// TIA Portal project "Ejercicio2_AutoGarbigailua" (V15.1)

(* hardware
DEVICE "S7-1200 station_1"  S7-1200 Station
   slot 0: "Rack_0"  S7-1200 Rack  Rack  V1.0
   slot 1: "PLC_1"  CPU 1214C AC/DC/Rly  6ES7 214-1BG40-0XB0  V4.2
*)

// ===== PLC "PLC_1"  CPU 1214C AC/DC/Rly =====

VAR_GLOBAL   // PLC tag table "Tabla de variables estándar"
   "Etapa4" AT %M16.4 : Bool;
   "Etapa3" AT %M16.3 : Bool;
   "Etapa2" AT %M16.2 : Bool;
   "Etapa1" AT %M16.1 : Bool;
   "Etapa0" AT %M16.0 : Bool;
   "S1" AT %I1.0 : Bool;
   "S2" AT %I1.1 : Bool;
   "S3" AT %I1.2 : Bool;
   "M" AT %I1.3 : Bool;
   "P" AT %I1.4 : Bool;
   "XV" AT %Q1.0 : Bool;
   "MP" AT %Q1.1 : Bool;
   "MC" AT %Q1.2 : Bool;
   "MV" AT %Q1.3 : Bool;
   "Etapa1.1" AT %M1.0 : Bool;
   "Etapa2.1" AT %M1.1 : Bool;
   "Etapa3.1" AT %M1.2 : Bool;
   "Etapa4.1" AT %M1.3 : Bool;
END_VAR

ORGANIZATION_BLOCK "Main"   // OB1, LAD, ProgramCycle
TITLE = "Main Program Sweep (Cycle)"
{ S7_Optimized_Access := 'TRUE' }
VERSION : 0.1
   VAR_INPUT
      Initial_Call : Bool;   // Initial call of this OB
      Remanence : Bool;   // =True, if remanent data are available
   END_VAR
   VAR_TEMP   // added for the SCL form of the ladder/FBD networks
      _w1 : Bool;
   END_VAR
BEGIN

REGION Network 1
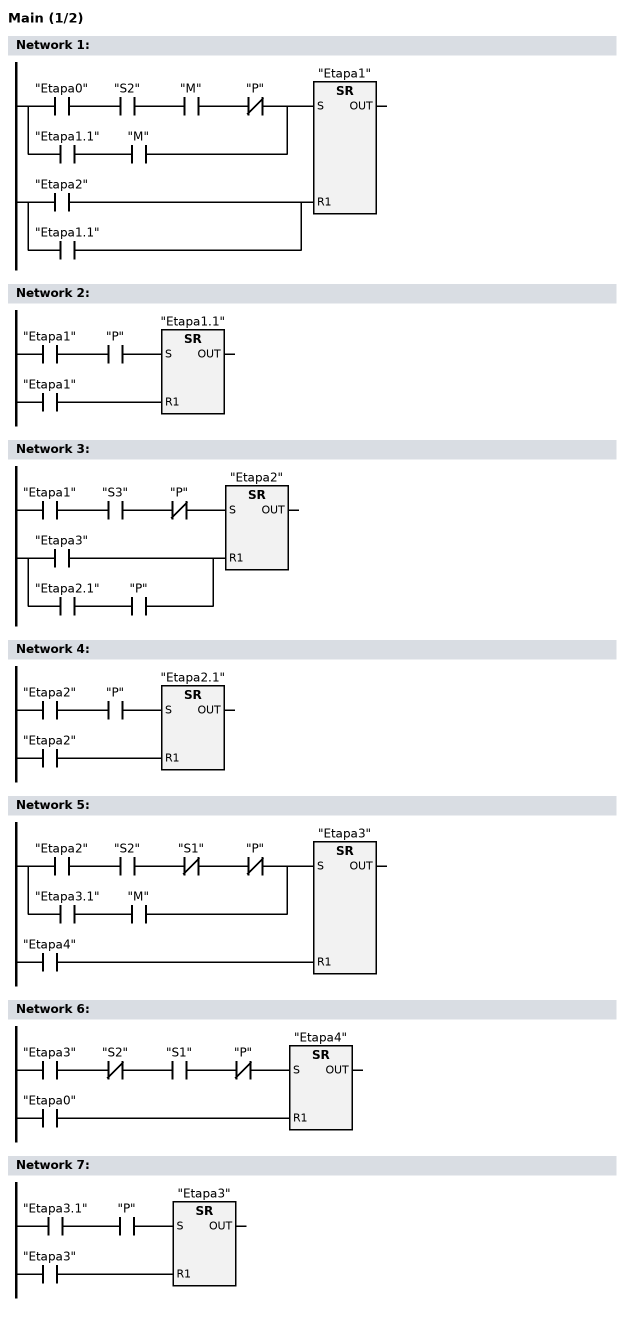
   RUNG wire#powerrail
      Contact( "Etapa0" )
      Contact( "S2" )
      Contact( "M" )
      I_Contact( "P" )
      wire#w1
      S_SR(operand := "Etapa1", r1 := wire#w2)
   END_RUNG
   RUNG wire#powerrail
      Contact( "Etapa1.1" )
      Contact( "M" )
   END_RUNG wire#w1
   RUNG wire#powerrail
      Contact( "Etapa2" )
   END_RUNG wire#w2
   RUNG wire#powerrail
      Contact( "Etapa1.1" )
   END_RUNG wire#w2
   // the same network as SCL:
   IF ("Etapa0" AND "S2" AND "M" AND NOT "P") OR ("Etapa1.1" AND "M") THEN
       "Etapa1" := TRUE;   // SR flip-flop
   END_IF;
   IF "Etapa2" OR "Etapa1.1" THEN "Etapa1" := FALSE; END_IF;
END_REGION

REGION Network 2
   RUNG wire#powerrail
      Contact( "Etapa1" )
      Contact( "P" )
      S_SR(operand := "Etapa1.1", r1 := wire#w1)
   END_RUNG
   RUNG wire#powerrail
      Contact( "Etapa1" )
   END_RUNG wire#w1
   // the same network as SCL:
   IF "Etapa1" AND "P" THEN
       "Etapa1.1" := TRUE;   // SR flip-flop
   END_IF;
   IF "Etapa1" THEN "Etapa1.1" := FALSE; END_IF;
END_REGION

REGION Network 3
   RUNG wire#powerrail
      Contact( "Etapa1" )
      Contact( "S3" )
      I_Contact( "P" )
      S_SR(operand := "Etapa2", r1 := wire#w1)
   END_RUNG
   RUNG wire#powerrail
      Contact( "Etapa3" )
   END_RUNG wire#w1
   RUNG wire#powerrail
      Contact( "Etapa2.1" )
      Contact( "P" )
   END_RUNG wire#w1
   // the same network as SCL:
   IF "Etapa1" AND "S3" AND NOT "P" THEN
       "Etapa2" := TRUE;   // SR flip-flop
   END_IF;
   IF "Etapa3" OR ("Etapa2.1" AND "P") THEN "Etapa2" := FALSE; END_IF;
END_REGION

REGION Network 4
   RUNG wire#powerrail
      Contact( "Etapa2" )
      Contact( "P" )
      S_SR(operand := "Etapa2.1", r1 := wire#w1)
   END_RUNG
   RUNG wire#powerrail
      Contact( "Etapa2" )
   END_RUNG wire#w1
   // the same network as SCL:
   IF "Etapa2" AND "P" THEN
       "Etapa2.1" := TRUE;   // SR flip-flop
   END_IF;
   IF "Etapa2" THEN "Etapa2.1" := FALSE; END_IF;
END_REGION

REGION Network 5
   RUNG wire#powerrail
      Contact( "Etapa2" )
      Contact( "S2" )
      I_Contact( "S1" )
      I_Contact( "P" )
      wire#w1
      S_SR(operand := "Etapa3", r1 := wire#w2)
   END_RUNG
   RUNG wire#powerrail
      Contact( "Etapa3.1" )
      Contact( "M" )
   END_RUNG wire#w1
   RUNG wire#powerrail
      Contact( "Etapa4" )
   END_RUNG wire#w2
   // the same network as SCL:
   IF ("Etapa2" AND "S2" AND NOT "S1" AND NOT "P") OR ("Etapa3.1" AND "M") THEN
       "Etapa3" := TRUE;   // SR flip-flop
   END_IF;
   IF "Etapa4" THEN "Etapa3" := FALSE; END_IF;
END_REGION

REGION Network 6
   RUNG wire#powerrail
      Contact( "Etapa3" )
      I_Contact( "S2" )
      Contact( "S1" )
      I_Contact( "P" )
      S_SR(operand := "Etapa4", r1 := wire#w1)
   END_RUNG
   RUNG wire#powerrail
      Contact( "Etapa0" )
   END_RUNG wire#w1
   // the same network as SCL:
   IF "Etapa3" AND NOT "S2" AND "S1" AND NOT "P" THEN
       "Etapa4" := TRUE;   // SR flip-flop
   END_IF;
   IF "Etapa0" THEN "Etapa4" := FALSE; END_IF;
END_REGION

REGION Network 7
   RUNG wire#powerrail
      Contact( "Etapa3.1" )
      Contact( "P" )
      S_SR(operand := "Etapa3", r1 := wire#w1)
   END_RUNG
   RUNG wire#powerrail
      Contact( "Etapa3" )
   END_RUNG wire#w1
   // the same network as SCL:
   #_w1 := "Etapa3";
   IF "Etapa3.1" AND "P" THEN
       "Etapa3" := TRUE;   // SR flip-flop
   END_IF;
   IF #_w1 THEN "Etapa3" := FALSE; END_IF;
END_REGION

REGION Network 8
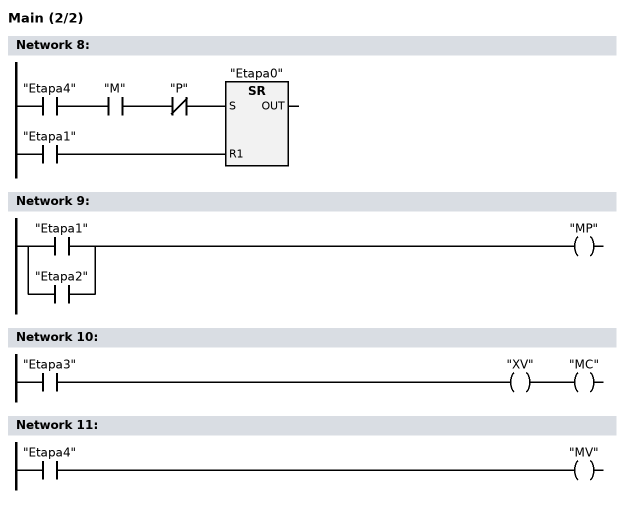
   RUNG wire#powerrail
      Contact( "Etapa4" )
      Contact( "M" )
      I_Contact( "P" )
      S_SR(operand := "Etapa0", r1 := wire#w1)
   END_RUNG
   RUNG wire#powerrail
      Contact( "Etapa1" )
   END_RUNG wire#w1
   // the same network as SCL:
   IF "Etapa4" AND "M" AND NOT "P" THEN
       "Etapa0" := TRUE;   // SR flip-flop
   END_IF;
   IF "Etapa1" THEN "Etapa0" := FALSE; END_IF;
END_REGION

REGION Network 9
   RUNG wire#powerrail
      Contact( "Etapa1" )
      wire#w1
      Coil( "MP" )
   END_RUNG
   RUNG wire#powerrail
      Contact( "Etapa2" )
   END_RUNG wire#w1
   // the same network as SCL:
   "MP" := "Etapa1" OR "Etapa2";
END_REGION

REGION Network 10
   RUNG wire#powerrail
      Contact( "Etapa3" )
      Coil( "XV" )
      Coil( "MC" )
   END_RUNG
   // the same network as SCL:
   "XV" := "Etapa3";
   "MC" := "Etapa3";
END_REGION

REGION Network 11
   RUNG wire#powerrail
      Contact( "Etapa4" )
      Coil( "MV" )
   END_RUNG
   // the same network as SCL:
   "MV" := "Etapa4";
END_REGION
END_ORGANIZATION_BLOCK

ORGANIZATION_BLOCK "Startup"   // OB100, LAD, Startup
TITLE = "Complete Restart"
{ S7_Optimized_Access := 'TRUE' }
VERSION : 0.1
   VAR_INPUT
      LostRetentive : Bool;   // True if retentive data are lost
      LostRTC : Bool;   // True if date and time are lost
   END_VAR
BEGIN

REGION Network 1
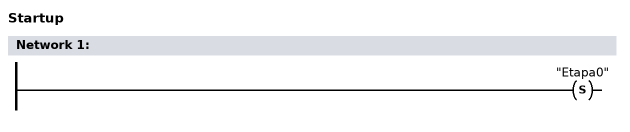
   RUNG wire#powerrail
      S_Coil( "Etapa0" )
   END_RUNG
   // the same network as SCL:
   "Etapa0" := TRUE;
END_REGION
END_ORGANIZATION_BLOCK